// TIA Portal V20 export
FUNCTION "06 T1-A ARUNC Output" : Void   // FC1602, LAD
TITLE = OUTPUT
{ S7_Optimized_Access := 'TRUE' }
// stored: AutoNumber false, SetENOAutomatically false
   VAR_TEMP
      Aux_real : Real;
      Aux_dint : DInt;
      Aux_uint : UInt;
      Aux_Bool : Bool;
      Aux_OS : Bool;
   END_VAR
BEGIN

REGION Network 1: ============= INTERLOCKS MOVING UP =============
END_REGION

REGION Network 2: Interlocks Move UP - Permanent Conditions
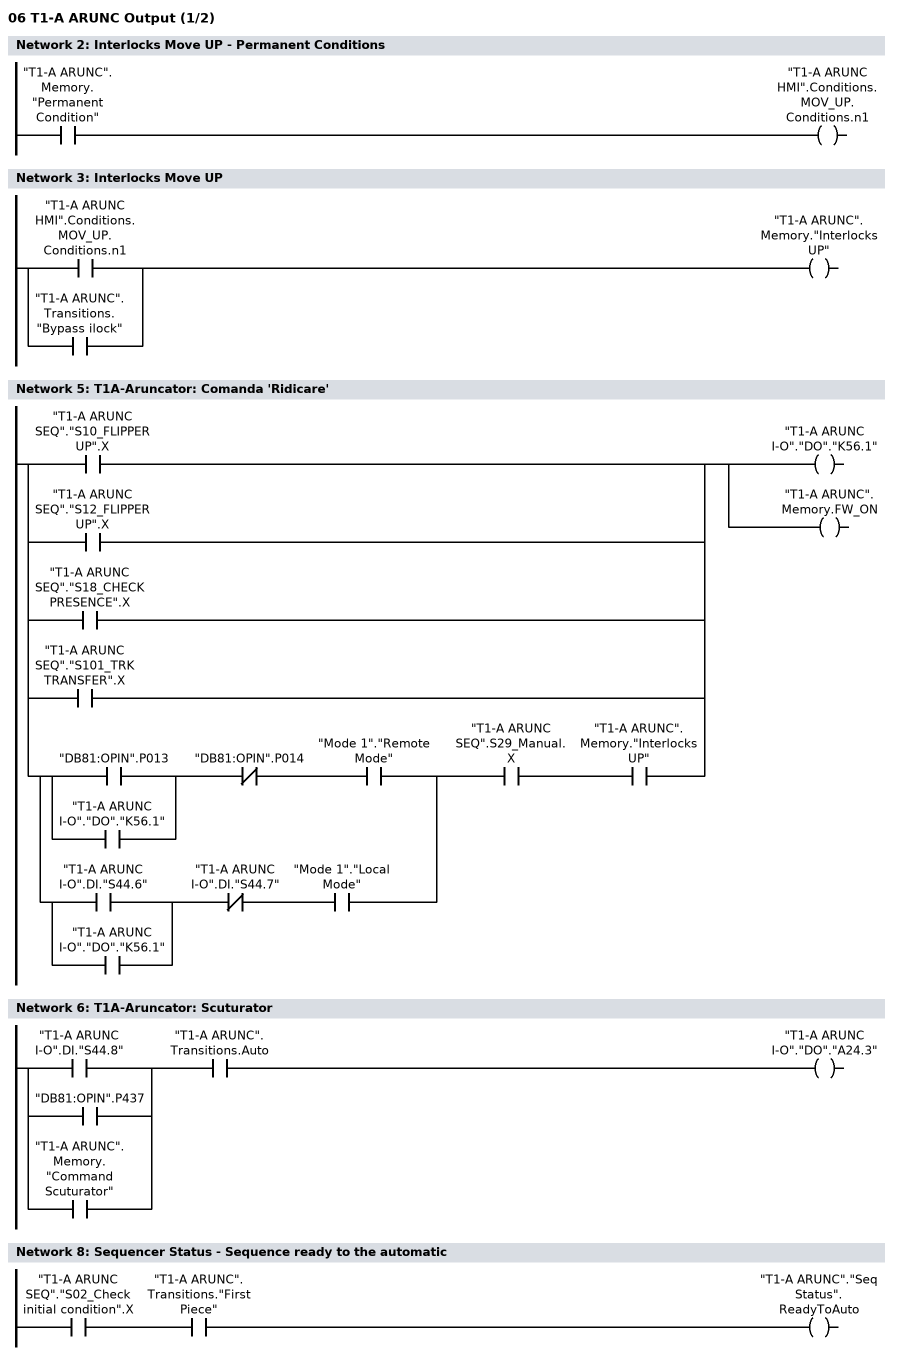
   RUNG wire#powerrail
      Contact( "T1-A ARUNC".Memory."Permanent Condition" )
      Coil( "T1-A ARUNC HMI".Conditions.MOV_UP.Conditions.n1 )
   END_RUNG
   // the same network as SCL:
   "T1-A ARUNC HMI".Conditions.MOV_UP.Conditions.n1 := "T1-A ARUNC".Memory."Permanent Condition";
END_REGION

REGION Network 3: Interlocks Move UP
   RUNG wire#powerrail
      Contact( "T1-A ARUNC HMI".Conditions.MOV_UP.Conditions.n1 )
      wire#w1
      Coil( "T1-A ARUNC".Memory."Interlocks UP" )
   END_RUNG
   RUNG wire#powerrail
      Contact( "T1-A ARUNC".Transitions."Bypass ilock" )
   END_RUNG wire#w1
   // the same network as SCL:
   "T1-A ARUNC".Memory."Interlocks UP" := "T1-A ARUNC HMI".Conditions.MOV_UP.Conditions.n1 OR "T1-A ARUNC".Transitions."Bypass ilock";
END_REGION

REGION Network 4: ============ COMMANDS ============
END_REGION

REGION Network 5: T1A-Aruncator: Comanda 'Ridicare'
   RUNG wire#powerrail
      Contact( "T1-A ARUNC SEQ"."S10_FLIPPER UP".X )
      wire#w1
      Coil( "T1-A ARUNC I-O"."DO"."K56.1" )
   END_RUNG
   RUNG wire#powerrail
      Contact( "T1-A ARUNC SEQ"."S12_FLIPPER UP".X )
   END_RUNG wire#w1
   RUNG wire#powerrail
      Contact( "T1-A ARUNC SEQ"."S18_CHECK PRESENCE".X )
   END_RUNG wire#w1
   RUNG wire#powerrail
      Contact( "T1-A ARUNC SEQ"."S101_TRK TRANSFER".X )
   END_RUNG wire#w1
   RUNG wire#powerrail
      Contact( "DB81:OPIN".P013 )
      wire#w2
      I_Contact( "DB81:OPIN".P014 )
      Contact( "Mode 1"."Remote Mode" )
      wire#w3
      Contact( "T1-A ARUNC SEQ".S29_Manual.X )
      Contact( "T1-A ARUNC".Memory."Interlocks UP" )
   END_RUNG wire#w1
   RUNG wire#powerrail
      Contact( "T1-A ARUNC I-O"."DO"."K56.1" )
   END_RUNG wire#w2
   RUNG wire#powerrail
      Contact( "T1-A ARUNC I-O".DI."S44.6" )
      wire#w4
      I_Contact( "T1-A ARUNC I-O".DI."S44.7" )
      Contact( "Mode 1"."Local Mode" )
   END_RUNG wire#w3
   RUNG wire#powerrail
      Contact( "T1-A ARUNC I-O"."DO"."K56.1" )
   END_RUNG wire#w4
   RUNG wire#w1
      Coil( "T1-A ARUNC".Memory.FW_ON )
   END_RUNG
   // the same network as SCL:
   "T1-A ARUNC I-O"."DO"."K56.1" := "T1-A ARUNC SEQ"."S10_FLIPPER UP".X OR "T1-A ARUNC SEQ"."S12_FLIPPER UP".X OR "T1-A ARUNC SEQ"."S18_CHECK PRESENCE".X OR "T1-A ARUNC SEQ"."S101_TRK TRANSFER".X OR (((("DB81:OPIN".P013 OR "T1-A ARUNC I-O"."DO"."K56.1") AND NOT "DB81:OPIN".P014 AND "Mode 1"."Remote Mode") OR (("T1-A ARUNC I-O".DI."S44.6" OR "T1-A ARUNC I-O"."DO"."K56.1") AND NOT "T1-A ARUNC I-O".DI."S44.7" AND "Mode 1"."Local Mode")) AND "T1-A ARUNC SEQ".S29_Manual.X AND "T1-A ARUNC".Memory."Interlocks UP");
   "T1-A ARUNC".Memory.FW_ON := "T1-A ARUNC I-O"."DO"."K56.1";
END_REGION

REGION Network 6: T1A-Aruncator: Scuturator
   RUNG wire#powerrail
      Contact( "T1-A ARUNC I-O".DI."S44.8" )
      wire#w1
      Contact( "T1-A ARUNC".Transitions.Auto )
      Coil( "T1-A ARUNC I-O"."DO"."A24.3" )
   END_RUNG
   RUNG wire#powerrail
      Contact( "DB81:OPIN".P437 )
   END_RUNG wire#w1
   RUNG wire#powerrail
      Contact( "T1-A ARUNC".Memory."Command Scuturator" )
   END_RUNG wire#w1
   // the same network as SCL:
   "T1-A ARUNC I-O"."DO"."A24.3" := ("T1-A ARUNC I-O".DI."S44.8" OR "DB81:OPIN".P437 OR "T1-A ARUNC".Memory."Command Scuturator") AND "T1-A ARUNC".Transitions.Auto;
END_REGION

REGION Network 7: ================== SEQUENCER STATUS ==================
END_REGION

REGION Network 8: Sequencer Status - Sequence ready to the automatic
   RUNG wire#powerrail
      Contact( "T1-A ARUNC SEQ"."S02_Check initial condition".X )
      Contact( "T1-A ARUNC".Transitions."First Piece" )
      Coil( "T1-A ARUNC"."Seq Status".ReadyToAuto )
   END_RUNG
   // the same network as SCL:
   "T1-A ARUNC"."Seq Status".ReadyToAuto := "T1-A ARUNC SEQ"."S02_Check initial condition".X AND "T1-A ARUNC".Transitions."First Piece";
END_REGION

REGION Network 9: Sequencer Status - Sequencer auto active
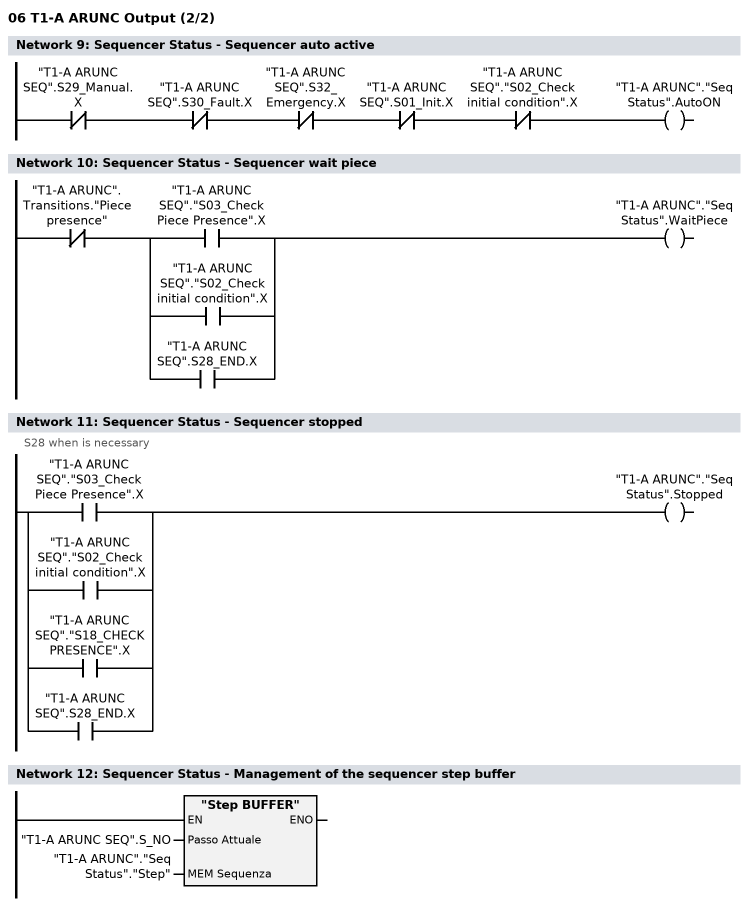
   RUNG wire#powerrail
      I_Contact( "T1-A ARUNC SEQ".S29_Manual.X )
      I_Contact( "T1-A ARUNC SEQ".S30_Fault.X )
      I_Contact( "T1-A ARUNC SEQ".S32_Emergency.X )
      I_Contact( "T1-A ARUNC SEQ".S01_Init.X )
      I_Contact( "T1-A ARUNC SEQ"."S02_Check initial condition".X )
      Coil( "T1-A ARUNC"."Seq Status".AutoON )
   END_RUNG
   // the same network as SCL:
   "T1-A ARUNC"."Seq Status".AutoON := NOT "T1-A ARUNC SEQ".S29_Manual.X AND NOT "T1-A ARUNC SEQ".S30_Fault.X AND NOT "T1-A ARUNC SEQ".S32_Emergency.X AND NOT "T1-A ARUNC SEQ".S01_Init.X AND NOT "T1-A ARUNC SEQ"."S02_Check initial condition".X;
END_REGION

REGION Network 10: Sequencer Status - Sequencer wait piece
   RUNG wire#powerrail
      I_Contact( "T1-A ARUNC".Transitions."Piece presence" )
      wire#w1
      Contact( "T1-A ARUNC SEQ"."S03_Check Piece Presence".X )
      wire#w2
      Coil( "T1-A ARUNC"."Seq Status".WaitPiece )
   END_RUNG
   RUNG wire#w1
      Contact( "T1-A ARUNC SEQ"."S02_Check initial condition".X )
   END_RUNG wire#w2
   RUNG wire#w1
      Contact( "T1-A ARUNC SEQ".S28_END.X )
   END_RUNG wire#w2
   // the same network as SCL:
   "T1-A ARUNC"."Seq Status".WaitPiece := NOT "T1-A ARUNC".Transitions."Piece presence" AND ("T1-A ARUNC SEQ"."S03_Check Piece Presence".X OR "T1-A ARUNC SEQ"."S02_Check initial condition".X OR "T1-A ARUNC SEQ".S28_END.X);
END_REGION

REGION Network 11: Sequencer Status - Sequencer stopped
   // S28 when is necessary
   RUNG wire#powerrail
      Contact( "T1-A ARUNC SEQ"."S03_Check Piece Presence".X )
      wire#w1
      Coil( "T1-A ARUNC"."Seq Status".Stopped )
   END_RUNG
   RUNG wire#powerrail
      Contact( "T1-A ARUNC SEQ"."S02_Check initial condition".X )
   END_RUNG wire#w1
   RUNG wire#powerrail
      Contact( "T1-A ARUNC SEQ"."S18_CHECK PRESENCE".X )
   END_RUNG wire#w1
   RUNG wire#powerrail
      Contact( "T1-A ARUNC SEQ".S28_END.X )
   END_RUNG wire#w1
   // the same network as SCL:
   "T1-A ARUNC"."Seq Status".Stopped := "T1-A ARUNC SEQ"."S03_Check Piece Presence".X OR "T1-A ARUNC SEQ"."S02_Check initial condition".X OR "T1-A ARUNC SEQ"."S18_CHECK PRESENCE".X OR "T1-A ARUNC SEQ".S28_END.X;
END_REGION

REGION Network 12: Sequencer Status - Management of the sequencer step buffer
   RUNG wire#powerrail
      "Step BUFFER"("Passo Attuale" := "T1-A ARUNC SEQ".S_NO, "MEM Sequenza" := "T1-A ARUNC"."Seq Status"."Step")
   END_RUNG
   // the same network as SCL:
   "Step BUFFER"("Passo Attuale" := "T1-A ARUNC SEQ".S_NO, "MEM Sequenza" := "T1-A ARUNC"."Seq Status"."Step");
END_REGION
END_FUNCTION
